{attribute addProperty BoxType "EJ1914-0000-0017"}
{attribute addProperty Id "EMPTY_STRUCTURE"}
{attribute addProperty CRC "0"}
{attribute addProperty SizeInBites "0"}
{attribute addProperty SizeInBytes "0"}
TYPE EMPTY_STRUCTURE :
STRUCT
END_STRUCT
END_TYPE

(* stored: Version 1.2.0.0, ProductVersion 3.1.4024.9
   DUT EMPTY_STRUCTURE: Id {996f7f70-7c97-40f1-8697-8e149ef8529e} *)
